(*
version 1.0	21 feb 2008
programmer 	hugo
tested by	oscat

this function add two complex numbers

*)
FUNCTION CADD : complex
VAR_INPUT
	X, Y : complex;
END_VAR

CADD.re := x.re + y.re;
CADD.im := x.im + y.im;


(* revision history
hm	21. feb 2008	rev 1.0
	original version

*)

END_FUNCTION

(* stored: Version 1.1.0.1
   POU CADD: Id {b012cf33-51cb-4efd-a354-0f7e80788406}, SpecialFunc None *)
